FUNCTION_BLOCK FB_FeedMeina2_500x500 EXTENDS FB_RecipeBase

METHOD Build : BOOL
VAR
    TotalX, TotalY, Radius : LREAL;
    Velo : LREAL;
    localConfig : ST_GantryXYZ_Config;
	
    // Zmienne do otworów
    HoleDistanceFromEdgeOfRail : LREAL := 100.0;
    SomeFixedDimension         : LREAL := 12.63;
    PanelRailOffsetX           : LREAL;
    PanelRailOffsetY           : LREAL;
    ExtrusionLengthX           : LREAL;
    ExtrusionLengthY           : LREAL;
    
    NumberOfHolesX             : INT := 3;
    NumberOfHolesY             : INT := 5;
    HolesSpacingX              : LREAL;
    HolesSpacingY              : LREAL;
    
    i                          : INT;
    holeIdx                    : INT;
	
	RailSlot  : LREAL := 29.0;
	BigSlot   : LREAL := 200.0;
	SmallSlot : LREAL := 100.0;

	PanelW : ARRAY[1..5] OF LREAL;
    PanelH : ARRAY[1..5] OF LREAL;
    PanelR : ARRAY[1..5] OF LREAL;
    X_Offset : LREAL;
    Y_Offset : LREAL;
    p : INT;

    // Stały wymiar szczelin ekstruzyjnych
    BaseExtrusion : LREAL;
	
	
// Zmienne pomocnicze do generowania ścieżek
	sx : LREAL;
	sy : LREAL;
	dx : LREAL;
	dy : LREAL;
	r_val : LREAL;
	
END_VAR
_Busy := TRUE;
_Done := FALSE;
_Error := FALSE;
Build := FALSE;
THIS^.UpdateNestingLimits();

IF NOT _Config.IsValid THEN
    _Busy := FALSE;
    _Error := TRUE; 
    Build := FALSE;
    RETURN;
END_IF

// ===================================================
// DEFINICJA PANELI GŁÓWNYCH (1 duży + 4 małe)
// ===================================================
// 1. Duży kwadrat (Oryginał)
_ShapeStart[1].X := 0.0;     _ShapeStart[1].Y := 0.0;
PanelW[1] := 1000.0;         PanelH[1] := 1000.0;
PanelR[1] := _Config.Radius; 

// 2. Mały kwadrat 1
_ShapeStart[2].X := 0.0;     _ShapeStart[2].Y := 1020.0;
PanelW[2] := 500.0;          PanelH[2] := 500.0;
PanelR[2] := 10.0;

// 3. Mały kwadrat 2
_ShapeStart[3].X := 0.0;     _ShapeStart[3].Y := 1540.0;
PanelW[3] := 500.0;          PanelH[3] := 500.0;
PanelR[3] := 10.0;

// 4. Mały kwadrat 3
_ShapeStart[4].X := 520.0;   _ShapeStart[4].Y := 1020.0;
PanelW[4] := 500.0;          PanelH[4] := 500.0;
PanelR[4] := 10.0;

// 5. Mały kwadrat 4
_ShapeStart[5].X := 520.0;   _ShapeStart[5].Y := 1540.0;
PanelW[5] := 500.0;          PanelH[5] := 500.0;
PanelR[5] := 10.0;

// ===================================================
// GENEROWANIE OTWORÓW DLA WSZYSTKICH 5 PANELI
// ===================================================
holeIdx := 0; 

FOR p := 1 TO 5 DO
    // Pobranie wymiarów dla aktualnie obliczanego panelu
    TotalX := PanelW[p];
    TotalY := PanelH[p];
    X_Offset := _ShapeStart[p].X;
    Y_Offset := _ShapeStart[p].Y;

    // Offsety i wyliczenia proporcjonalne do wymiarów konkretnego panelu
    PanelRailOffsetX := 0.1 * TotalX;
    PanelRailOffsetY := 0.1 * TotalY;

    ExtrusionLengthX := TotalX - (2.0 * PanelRailOffsetX);
    ExtrusionLengthY := TotalY - (2.0 * PanelRailOffsetY);

    IF NumberOfHolesX > 1 THEN
        HolesSpacingX := (ExtrusionLengthX - (2.0 * HoleDistanceFromEdgeOfRail)) / INT_TO_LREAL(NumberOfHolesX - 1);
    ELSE
        HolesSpacingX := 0.0;
    END_IF

    IF NumberOfHolesY > 1 THEN
        HolesSpacingY := (ExtrusionLengthY - (2.0 * HoleDistanceFromEdgeOfRail)) / INT_TO_LREAL(NumberOfHolesY - 1);
    ELSE
        HolesSpacingY := 0.0;
    END_IF

    // 1. Otwór na środku danego panelu
    holeIdx := holeIdx + 1;
    _HolesDrill[holeIdx].X := LREAL_TO_REAL((TotalX / 2.0) + X_Offset);
    _HolesDrill[holeIdx].Y := LREAL_TO_REAL((TotalY / 2.0) + Y_Offset);

    // 2. Rail Y1 (Lewa)
    FOR i := NumberOfHolesY TO 1 BY -1 DO
        holeIdx := holeIdx + 1;
        _HolesDrill[holeIdx].X := LREAL_TO_REAL(PanelRailOffsetX - SomeFixedDimension + X_Offset);
        _HolesDrill[holeIdx].Y := LREAL_TO_REAL(PanelRailOffsetY + HoleDistanceFromEdgeOfRail + ((i - 1) * HolesSpacingY) + Y_Offset);
    END_FOR

    // 3. Rail X1 (Dolna)
    FOR i := 1 TO NumberOfHolesX DO
        holeIdx := holeIdx + 1;
        _HolesDrill[holeIdx].X := LREAL_TO_REAL(PanelRailOffsetX + HoleDistanceFromEdgeOfRail + ((i - 1) * HolesSpacingX) + X_Offset);
        _HolesDrill[holeIdx].Y := LREAL_TO_REAL(PanelRailOffsetY - SomeFixedDimension + Y_Offset);
    END_FOR

    // 4. Rail Y2 (Prawa)
    FOR i := 1 TO NumberOfHolesY DO
        holeIdx := holeIdx + 1;
        _HolesDrill[holeIdx].X := LREAL_TO_REAL(PanelRailOffsetX + ExtrusionLengthX + SomeFixedDimension + X_Offset);
        _HolesDrill[holeIdx].Y := LREAL_TO_REAL(PanelRailOffsetY + HoleDistanceFromEdgeOfRail + ((i - 1) * HolesSpacingY) + Y_Offset);
    END_FOR

    // 5. Rail X2 (Górna)
    FOR i := NumberOfHolesX TO 1 BY -1 DO
        holeIdx := holeIdx + 1;
        _HolesDrill[holeIdx].X := LREAL_TO_REAL(PanelRailOffsetX + HoleDistanceFromEdgeOfRail + ((i - 1) * HolesSpacingX) + X_Offset);
        _HolesDrill[holeIdx].Y := LREAL_TO_REAL(PanelRailOffsetY + ExtrusionLengthY + SomeFixedDimension + Y_Offset);
    END_FOR
END_FOR

_HolesToDrill := holeIdx;

// ===================================================
// POZOSTAŁE WYCIĘCIA
// ===================================================
_ShapesCount := 10; // 5 paneli głównych + 5 małych wycięć

// No. 1 do No. 5 z poprzednich ustawień
_ShapeStart[6].X := 1030.0; _ShapeStart[6].Y := 0.0;
_ShapeStart[7].X := 1090.0; _ShapeStart[7].Y := 0.0;
_ShapeStart[8].X := 210.0;  _ShapeStart[8].Y := 2200.0;
_ShapeStart[9].X := 410.0;  _ShapeStart[9].Y := 2150.0;
_ShapeStart[10].X := 810.0; _ShapeStart[10].Y := 2150.0;

IF _ConfigProvider <> 0 THEN
    localConfig := _ConfigProvider.Config;
    Velo := localConfig.CuttingSpeedXY;
ELSE
    Velo := 50.0;
END_IF

_GeometryWriter.Clear();
_GeometryWriter.EnableTangentialFollowing();

sx := 0.0; sy := 0.0; dx := 0.0; dy := 0.0; r_val := 0.0;

// RYSOWANIE KSZTAŁTU ZGODNIE Z INDEKSEM
CASE _CurrentShapeIndex OF
    1, 2, 3, 4, 5:
        // ==========================================
        // RYSOWANIE PANELI (1 Duży + 4 Małe)
        // ==========================================
        sx := _ShapeStart[_CurrentShapeIndex].X;
        sy := _ShapeStart[_CurrentShapeIndex].Y;
        TotalX := PanelW[_CurrentShapeIndex];
        TotalY := PanelH[_CurrentShapeIndex];
        Radius := PanelR[_CurrentShapeIndex];

        IF Radius > (TotalX / 2.0) THEN Radius := TotalX / 2.0; END_IF
        IF Radius > (TotalY / 2.0) THEN Radius := TotalY / 2.0; END_IF

        _GeometryWriter.AddStartPoint(sx, sy);

        _GeometryWriter.AddLine(sx, sy + TotalY - Radius, Velo);
        IF Radius > 0 THEN
            _GeometryWriter.AddArc(sx + Radius, sy + TotalY, sx + Radius, sy + TotalY - Radius, Velo, TRUE);
        END_IF

        _GeometryWriter.AddLine(sx + TotalX - Radius, sy + TotalY, Velo);
        IF Radius > 0 THEN
            _GeometryWriter.AddArc(sx + TotalX, sy + TotalY - Radius, sx + TotalX - Radius, sy + TotalY - Radius, Velo, TRUE);
        END_IF

        _GeometryWriter.AddLine(sx + TotalX, sy + Radius, Velo);
        IF Radius > 0 THEN
            _GeometryWriter.AddArc(sx + TotalX - Radius, sy, sx + TotalX - Radius, sy + Radius, Velo, TRUE);
        END_IF

        _GeometryWriter.AddLine(sx + Radius, sy, Velo);
        IF Radius > 0 THEN
            _GeometryWriter.AddArc(sx, sy + Radius, sx + Radius, sy + Radius, Velo, TRUE);
        END_IF

    6, 7, 8, 9, 10:
        // ==========================================
        // RYSOWANIE WYCIĘĆ NA PROFILE
        // ==========================================
        sx := _ShapeStart[_CurrentShapeIndex].X;
        sy := _ShapeStart[_CurrentShapeIndex].Y;
        r_val := 10.0;

        // Stały wymiar dy/dx oparty na panelu 1000x1000: 1000 - 2*(10% z 1000) = 800
        BaseExtrusion := 800.0; 

        IF _CurrentShapeIndex = 6 THEN
            dx := RailSlot;
            dy := BaseExtrusion;
        ELSIF _CurrentShapeIndex = 7 THEN
            dx := RailSlot;
            dy := BaseExtrusion; 
        ELSIF _CurrentShapeIndex = 8 THEN
            dx := SmallSlot;
            dy := SmallSlot;
        ELSIF _CurrentShapeIndex = 9 THEN
            dx := BigSlot;
            dy := BigSlot;
        ELSIF _CurrentShapeIndex = 10 THEN
            dx := BigSlot;
            dy := BigSlot;
        END_IF

        _GeometryWriter.AddStartPoint(sx, sy);

        _GeometryWriter.AddLine(sx, sy + dy - r_val, Velo);
        IF r_val > 0 THEN
            _GeometryWriter.AddArc(sx + r_val, sy + dy, sx + r_val, sy + dy - r_val, Velo, TRUE);
        END_IF

        _GeometryWriter.AddLine(sx + dx - r_val, sy + dy, Velo);
        IF r_val > 0 THEN
            _GeometryWriter.AddArc(sx + dx, sy + dy - r_val, sx + dx - r_val, sy + dy - r_val, Velo, TRUE);
        END_IF

        _GeometryWriter.AddLine(sx + dx, sy + r_val, Velo);
        IF r_val > 0 THEN
            _GeometryWriter.AddArc(sx + dx - r_val, sy, sx + dx - r_val, sy + r_val, Velo, TRUE);
        END_IF

        _GeometryWriter.AddLine(sx + r_val, sy, Velo);
        IF r_val > 0 THEN
            _GeometryWriter.AddArc(sx, sy + r_val, sx + r_val, sy + r_val, Velo, TRUE);
        END_IF

END_CASE

_GeometryWriter.EndTable();

_Busy := FALSE;
_Done := TRUE;
Build := TRUE;
END_METHOD

METHOD PROTECTED CalculateFootprint
VAR_INPUT
END_VAR
_NominalX := 1200;
_NominalY := 2400;
END_METHOD

PROPERTY ExecutionRoute : E_ExecutionRoute
GET
ExecutionRoute := E_ExecutionRoute.eFeedTable;
END_GET
END_PROPERTY

METHOD FB_init : BOOL
VAR_INPUT
	bInitRetains : BOOL; // if TRUE, the retain variables are initialized (warm start / cold start)
	bInCopyCode : BOOL;  // if TRUE, the instance afterwards gets moved into the copy code (online change)
END_VAR
_Limits.PanelFrontLength.MinVal := 100.0;
_Limits.PanelFrontLength.MaxVal := 2400.0;

_Limits.PanelFrontWidth.MinVal  := 100.0;
_Limits.PanelFrontWidth.MaxVal  := 1200.0;

_Limits.PanelHeight.MinVal      := 0.0;
_Limits.PanelHeight.MaxVal      := 0.0;

_Limits.RailHeightCorrection.MinVal := 0.0;
_Limits.RailHeightCorrection.MaxVal := 0.0;

_Limits.CuttingOverpass.MinVal := 0.0;
_Limits.CuttingOverpass.MaxVal := 50.0;

_Limits.GroovingOverpass.MinVal := 0.0;
_Limits.GroovingOverpass.MaxVal := 50.0;

_Limits.GrooveDepthZ.MinVal := 0.0;
_Limits.GrooveDepthZ.MaxVal := 9.0; 

_Limits.CuttingOverpass.MinVal := 0.0;
_Limits.CuttingOverpass.MaxVal := 50.0;
_Limits.GroovingOverpass.MinVal := 0.0;
_Limits.GroovingOverpass.MaxVal := 50.0;

_Limits.Radius.MinVal := 10.0;     
_Limits.Radius.MaxVal := 600.0;
END_METHOD

END_FUNCTION_BLOCK

(* stored: Version 1.1.0.1, ProductVersion 3.1.4024.15
   POU FB_FeedMeina2_500x500: Id {55576838-7eac-41b8-bcab-a7bf7fbec968}, SpecialFunc None
   Method Build: Id {dfa8aa9e-d1ba-4342-be9a-7fd13ab5c17a}
   Method CalculateFootprint: Id {51ef9402-89b9-4a0f-aa8f-6c97ea01621c}
   Property ExecutionRoute: Id {769e0bae-c163-4201-a397-e4a11e8f8fed}
   Get Get: Id {43526d1a-f06a-41e1-b46f-a5df63c0d3fc}
   Method FB_init: Id {daa1d0e9-b1d9-4e64-a410-5a60a0bc6389} *)
